Universal Robots PolyScope program: move_on_grid.urp

Program move_on_grid (installation=default directory=/programs/DND createdIn=5.12.4.1101661 lastSavedIn=5.12.4.1101661 robotSerialNumber=20225502378)
Calibrated DH parameters: a=[0.00022, -0.425328, -0.389701, 0.000059, 0.000065, 0]; d=[0.162608, 0.803456, 9.992211, -10.662202, 0.099702, 0.099559]; alpha=[1.570756, 0.001543, 0.004316, 1.570651, -1.570122, 0]; deltaTheta=[0, 0.002917, 0.116094, -0.119008, 0, -0.000001]
Robot Program (runOnlyOnce=true)
  tile_pos_id := GP_int_in[0]
  grid_pos_id := GP_int_in[1]
  ter_hover_pos := p[0,0,0,0,0,0]
  ter_lower_pos := p[0, 0, 0, 0, 0, 0]
  grid_hover_pos := p[0,0,0,0,0,0]
  grid_lower_pos := p[0,0,0,0,0,0]
  Script file /programs/DND/hov_offset_calc.script_bak
    | # Tile spacing
    | tile_spacing_x_ter = 0.091
    | tile_spacing_y_ter = 0.091
    | tile_spacing_x_grid = 0.0875
    | tile_spacing_y_grid =0.0875
    | 
    | #Extract Tile Row and Column for Chosen Terrain Tile
    | ter_tile_row = (floor(tile_pos_id / 10)) - 1
    | ter_tile_col = (tile_pos_id % 10) - 1
    | 
    | # Extract Row and Column for Target Grid Position
    | grid_tile_row = (floor(grid_pos_id / 10)) - 1
    | grid_tile_col = (grid_pos_id % 10) - 1
    | 
    | # Calculate Offset Poses
    | ter_hover_offset = p[-tile_spacing_x_ter * ter_tile_row, -tile_spacing_y_ter * ter_tile_col, 0, 0, 0, 0]
    | grid_hover_offset = p[-tile_spacing_x_grid * grid_tile_row, -tile_spacing_y_grid * grid_tile_col, 0, 0, 0, 0]
    | 
    | # Calculate Final Pos
    | ter_hover_pos = pose_add(ter_base_hover, ter_hover_offset)
    | ter_lower_pos = pose_add(ter_hover_pos, p[0,0,-0.109,0,0,0])
    | grid_hover_pos = pose_add(grid_base_hover, grid_hover_offset)
    | grid_lower_pos = pose_add(grid_hover_pos, p[0,0,-0.079,0,0,0])
  MoveL speed 250 mm/s, acceleration 1200 mm/s^2 (useActiveTCP=true) feature=Base
    Waypoint Waypoint (Variable): variable=ter_hover_pos
  URCap Gripper (Robotiq_Grippers, Robotiq Inc.) dataModel(position=75.0, force=0.0, speed=0.0, positionInDouble=75.0, forceInDouble=0.0, speedInDouble=0.0, slaveIds=[9], blocking=true)
  MoveL speed 250 mm/s, acceleration 1200 mm/s^2 (useActiveTCP=true) feature=Base
    Waypoint Waypoint (Variable): variable=ter_lower_pos
  URCap Gripper (Robotiq_Grippers, Robotiq Inc.) dataModel(position=100.0, force=0.0, speed=0.0, positionInDouble=100.0, forceInDouble=0.0, speedInDouble=0.0, slaveIds=[9], blocking=true)
  MoveL speed 250 mm/s, acceleration 1200 mm/s^2 (useActiveTCP=true) feature=Base
    Waypoint Waypoint (Variable): variable=ter_hover_pos
  MoveJ speed 60 deg/s, acceleration 80 deg/s^2 (useActiveTCP=true) feature=Base
    Waypoint Waypoint (Variable): variable=grid_hover_pos
  MoveL speed 250 mm/s, acceleration 1200 mm/s^2 (useActiveTCP=true) feature=Base
    Waypoint Waypoint (Variable): variable=grid_lower_pos
  URCap Gripper (Robotiq_Grippers, Robotiq Inc.) dataModel(position=75.0, force=0.0, speed=0.0, positionInDouble=75.0, forceInDouble=0.0, speedInDouble=0.0, slaveIds=[9], blocking=true)
  MoveL speed 250 mm/s, acceleration 1200 mm/s^2 (useActiveTCP=true) feature=Base
    Waypoint Waypoint (Variable): variable=grid_hover_pos
  URCap Gripper (Robotiq_Grippers, Robotiq Inc.) dataModel(position=74.90196078431373, force=0.0, speed=0.0, positionInDouble=74.90196078431373, forceInDouble=0.0, speedInDouble=0.0, slaveIds=[9], blocking=true)
  MoveL speed 250 mm/s, acceleration 1200 mm/s^2 (useActiveTCP=true) feature=Base
    Waypoint Waypoint (Variable): variable=grid_base_hover
